{attribute 'qualified_only'}
{attribute 'strict'}
TYPE E_CoordinatesSortState :
(
	eCoordinatesSortState_undefined := 0,
	eCoordinatesSortState_unsorted := 1,
	eCoordinatesSortState_sorted := 2,
	eCoordinatesSortState_resorted_v1 := 3
);
END_TYPE

(* stored: Version 1.1.0.1, ProductVersion 3.1.4022.9
   EnumerationTextList E_CoordinatesSortState: Id {60f7639d-0471-42a6-84be-a2a39d25dfb1} *)
